TYPE ZDataConfig :
STRUCT
{attribute '__ZwPlcApplicationDataConfigDeclaration__'} // Do not remove this attribute! It is used for code generation.
END_STRUCT
END_TYPE

(* stored: Version 1.1.0.1
   DUT ZDataConfig: Id {0b87d352-c0ca-4d72-a034-0b536674cab3} *)
